INTERFACE ITF_HMIManagerConfigure EXTENDS ITF_Base

METHOD PUBLIC SetActiveButtonMainMenu : BOOL
VAR_INPUT
	iButton			: INT;	//numer przycisku od 0
	bValue			: BOOL;	//true aktywny może być tylko jeden w menu
END_VAR
END_METHOD

METHOD PUBLIC SetEnableButtonMainMenu : BOOL
VAR_INPUT
	iButton			: INT;	//numer przycisku od 0
	bValue			: BOOL;	//true włączony
END_VAR
END_METHOD

METHOD PUBLIC SetVisibleButtonMainMenu : BOOL
VAR_INPUT
	iButton			: INT;	//numer przycisku od 0
	bValue			: BOOL;	//true widoczny
END_VAR
END_METHOD

END_INTERFACE

(* stored: Version 1.1.0.1
   Itf ITF_HMIManagerConfigure: Id {6d65f736-9707-03a5-294a-a8aaa4bb0d85}
   Method SetActiveButtonMainMenu: Id {4dd734d3-5e2a-057b-358d-afee9409412b}
   Method SetEnableButtonMainMenu: Id {9306a453-79bc-09ac-29a7-df180b99e765}
   Method SetVisibleButtonMainMenu: Id {ebe30521-ad78-08e6-2f96-9b2742b37c55} *)
